% RSLogix 500 project I2P JOB 12 B - SOLUTION.RSS, saved by version 10.00.00.00 %
PROJECT "UNTITLED"    % processor: Bul.1763 MicroLogix 1100 Series B %

PROGRAM FILES
  LAD 2   10 rungs

DATA FILES
  O0 OUTPUT  4 elements
  I1 INPUT  6 elements
  S2 STATUS  66 elements
  B3 BINARY  1 elements
  T4 TIMER  1 elements
  C5 COUNTER  1 elements
  R6 CONTROL  1 elements
  N7 INTEGER  1 elements
  F8 FLOAT  1 elements

LADDER 2
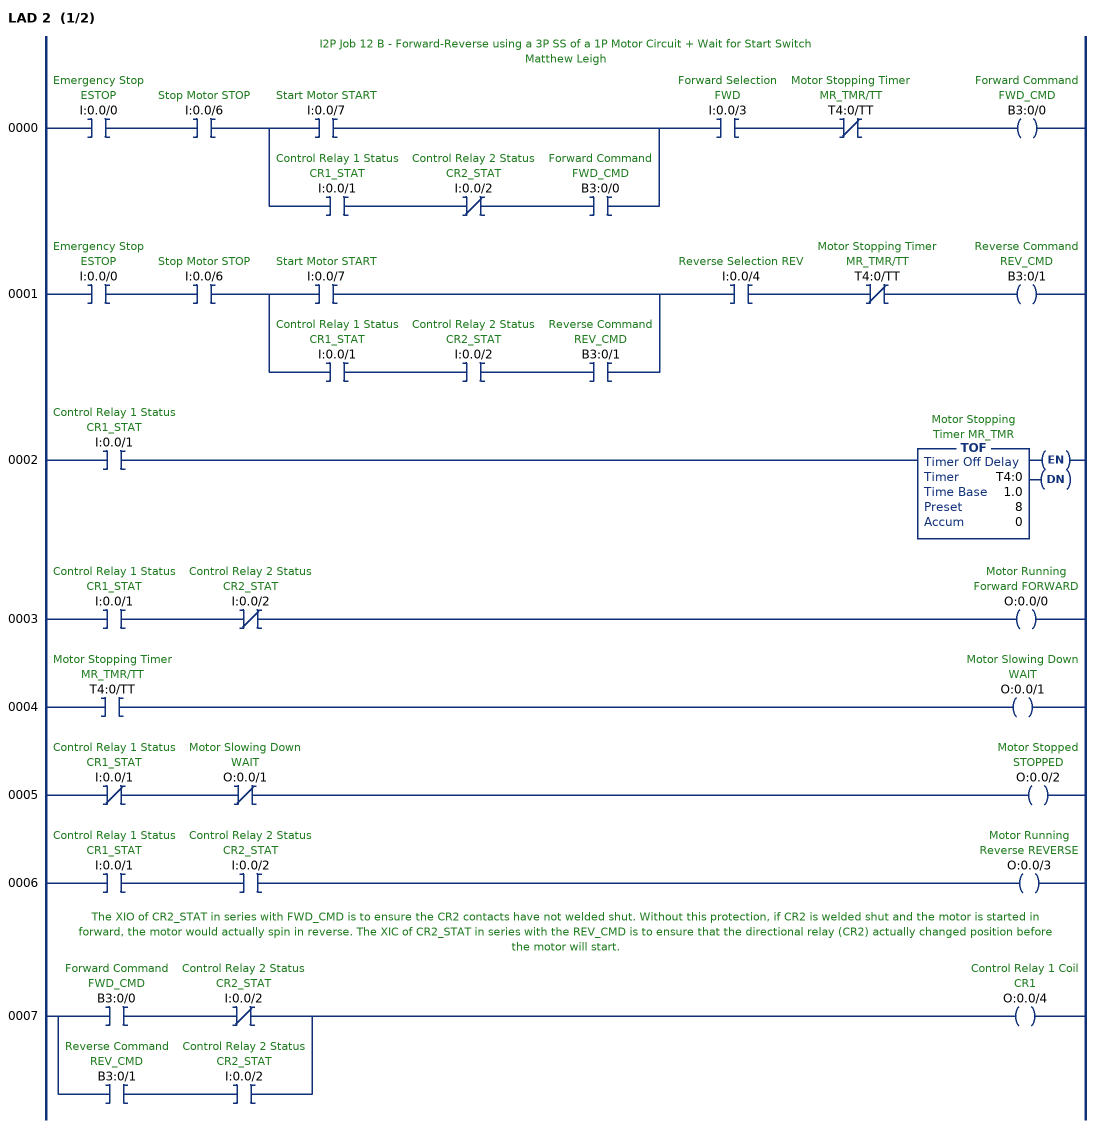
% Rung: 0 %
% I2P Job 12 B - Forward-Reverse using a 3P SS of a 1P Motor Circuit + Wait for Start Switch
% Matthew Leigh %
SOR XIC I:0.0/0 XIC I:0.0/6 BST XIC I:0.0/7 NXB XIC I:0.0/1 XIO I:0.0/2 XIC B3:0/0 BND XIC I:0.0/3 XIO T4:0/TT OTE B3:0/0 EOR
%   I:0.0/0  ESTOP  "Emergency Stop" %
%   I:0.0/6  STOP  "Stop Motor" %
%   I:0.0/7  START  "Start Motor" %
%   I:0.0/1  CR1_STAT  "Control Relay 1 Status" %
%   I:0.0/2  CR2_STAT  "Control Relay 2 Status" %
%   B3:0/0  FWD_CMD  "Forward Command" %
%   I:0.0/3  FWD  "Forward Selection" %
%   T4:0  MR_TMR  "Motor Stopping Timer" %
% Rung: 1 %
SOR XIC I:0.0/0 XIC I:0.0/6 BST XIC I:0.0/7 NXB XIC I:0.0/1 XIC I:0.0/2 XIC B3:0/1 BND XIC I:0.0/4 XIO T4:0/TT OTE B3:0/1 EOR
%   I:0.0/0  ESTOP  "Emergency Stop" %
%   I:0.0/6  STOP  "Stop Motor" %
%   I:0.0/7  START  "Start Motor" %
%   I:0.0/1  CR1_STAT  "Control Relay 1 Status" %
%   I:0.0/2  CR2_STAT  "Control Relay 2 Status" %
%   B3:0/1  REV_CMD  "Reverse Command" %
%   I:0.0/4  REV  "Reverse Selection" %
%   T4:0  MR_TMR  "Motor Stopping Timer" %
% Rung: 2 %
SOR XIC I:0.0/1 TOF T4:0 1.0 8 0 EOR
%   I:0.0/1  CR1_STAT  "Control Relay 1 Status" %
%   T4:0  MR_TMR  "Motor Stopping Timer" %
% Rung: 3 %
SOR XIC I:0.0/1 XIO I:0.0/2 OTE O:0.0/0 EOR
%   I:0.0/1  CR1_STAT  "Control Relay 1 Status" %
%   I:0.0/2  CR2_STAT  "Control Relay 2 Status" %
%   O:0.0/0  FORWARD  "Motor Running Forward" %
% Rung: 4 %
SOR XIC T4:0/TT OTE O:0.0/1 EOR
%   T4:0  MR_TMR  "Motor Stopping Timer" %
%   O:0.0/1  WAIT  "Motor Slowing Down" %
% Rung: 5 %
SOR XIO I:0.0/1 XIO O:0.0/1 OTE O:0.0/2 EOR
%   I:0.0/1  CR1_STAT  "Control Relay 1 Status" %
%   O:0.0/1  WAIT  "Motor Slowing Down" %
%   O:0.0/2  STOPPED  "Motor Stopped" %
% Rung: 6 %
SOR XIC I:0.0/1 XIC I:0.0/2 OTE O:0.0/3 EOR
%   I:0.0/1  CR1_STAT  "Control Relay 1 Status" %
%   I:0.0/2  CR2_STAT  "Control Relay 2 Status" %
%   O:0.0/3  REVERSE  "Motor Running Reverse" %
% Rung: 7 %
% The XIO of CR2_STAT in series with FWD_CMD is to ensure the CR2 contacts have not welded shut. Without this protection, if CR2 is welded shut and the motor is started in forward, the motor would actually spin in reverse. The XIC of CR2_STAT in series with the REV_CMD is to ensure that the directional relay (CR2) actually changed position before the motor will start. %
SOR BST XIC B3:0/0 XIO I:0.0/2 NXB XIC B3:0/1 XIC I:0.0/2 BND OTE O:0.0/4 EOR
%   B3:0/0  FWD_CMD  "Forward Command" %
%   I:0.0/2  CR2_STAT  "Control Relay 2 Status" %
%   B3:0/1  REV_CMD  "Reverse Command" %
%   O:0.0/4  CR1  "Control Relay 1 Coil" %

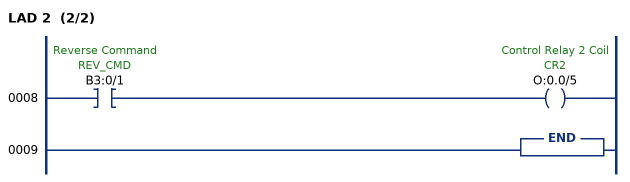
% Rung: 8 %
SOR XIC B3:0/1 OTE O:0.0/5 EOR
%   B3:0/1  REV_CMD  "Reverse Command" %
%   O:0.0/5  CR2  "Control Relay 2 Coil" %
% Rung: 9 %
SOR END EOR

OTHER DOCUMENTED ADDRESSES
  I:0.0/5  MODE  "Run/Jog Selector A=Run(1) & B=Jog(0)"
  I:0.0/8  JOG  "Jog Motor"

DATA TABLE (non-zero values as saved)
DATA T4
% .PRE .ACC %
% T4:0 % 8 0
